Staubli VAL3: find.pgx

public program find(string& x_sItem[], bool& x_bFound[])
  local num i
  local num l_nSize
  local string l_sEvent
begin
  // search a  SUB program
  // check if the item has been found
  x_bFound=isDefined(saveProg:pProg[x_sItem])
end
